GLOBALCONSTANTS SoftKeyActivationCode (* SoftKeyActivationCode constants *)
  (* Standard: 61499-1; Description: Copyright (c) 2024 HR Agrartechnik GmbH This program and the accompanying materials are made available under the terms of the Eclipse Public License 2.0 which is available at https://www.eclipse.org/legal/epl-2.0/ SPDX-License-Identifier: EPL-2.0 *)
  (* Version 1.0, 2024-01-25, Franz Höpfinger, HR Agrartechnik GmbH *)
  PACKAGE isobus::UT::io::Softkey;
  VAR_GLOBAL CONSTANT
    SK_RELEASED : isobus::UT::io::Softkey::SoftKeyActivationCode_S := (code := 0); (* SoftKey has been released (state change) *)
    SK_PRESSED : isobus::UT::io::Softkey::SoftKeyActivationCode_S := (code := 1); (* SoftKey  has been pressed (state change) *)
    SK_STILL_HELD : isobus::UT::io::Softkey::SoftKeyActivationCode_S := (code := 2); (* SoftKey is still held *)
    SK_STILL_HELD_START : isobus::UT::io::Softkey::SoftKeyActivationCode_S := (code := 2, bCyclic := FALSE); (* SoftKey is still held start *)
    SK_ABORTED : isobus::UT::io::Softkey::SoftKeyActivationCode_S := (code := 3); (* SoftKey press aborted (Applies to VT version 4 and later) *)
    Invalid : isobus::UT::io::Softkey::SoftKeyActivationCode_S := (code := 255);
  END_VAR
END_GLOBALCONSTANTS
